{attribute addProperty BoxType "BK1150-0000-0019"}
{attribute addProperty Id "Term_386_KL1002KL1002_D229A9CA00"}
{attribute addProperty CRC "2313591478"}
{attribute addProperty SizeInBites "0"}
{attribute addProperty SizeInBytes "0"}
TYPE A_0013_BK1150_0000_0019_89E69AB6 EXTENDS BK1150_A5F67C82 :
STRUCT
	{attribute addProperty Name "Term_386_KL1002"}
	Term_386_KL1002 : KL1002_D229A9CA;
END_STRUCT
END_TYPE

(* stored: Version 1.2.0.0, ProductVersion 3.1.4024.9
   DUT A_0013_BK1150_0000_0019_89E69AB6: Id {592dda9e-5c8d-4e15-b13e-bb90a1e4c20b} *)
